FUNCTION_BLOCK FB_TimeDelta
VAR
	StartTime : ST_TimeStruct;
    StopTime : ST_TimeStruct;
    CurrentTime : ST_TimeStruct; // Assuming this to be cyclically updated to the current PLC time
	fbGetSystemTime : GETSYSTEMTIME;
    timeAsFileTime : T_FILETIME;
    timeAsDT : DATE_AND_TIME;
END_VAR

F_GetSystemTime(F_GetSystemTime => CurrentTime);
GetDelta();

METHOD GetDelta : ST_TimeStruct
VAR
	DeltaTime : ST_TimeStruct;
	DaysInMonth : ARRAY[0..12] OF WORD := [0,31,28,31,30,31,30,31,31,30,31,30,31]; // Days in each month
	bLeapYear : BOOL;
END_VAR
// Calculate the delta TIME here AND assign it TO DeltaTime
	DeltaTime.wYear := StopTime.wYear - StartTime.wYear;
    DeltaTime.wMonth := StopTime.wMonth - StartTime.wMonth;
    DeltaTime.wDay := StopTime.wDay - StartTime.wDay;
    DeltaTime.wHour := StopTime.wHour - StartTime.wHour;
    DeltaTime.wMinute := StopTime.wMinute - StartTime.wMinute;
    DeltaTime.wSecond := StopTime.wSecond - StartTime.wSecond;
    DeltaTime.wMilliseconds := StopTime.wMilliseconds - StartTime.wMilliseconds;
	
// Calculate delta time
    IF StartTime.wMilliseconds > StopTime.wMilliseconds THEN
        DeltaTime.wMilliseconds := 65535 - DeltaTime.wMilliseconds;
    END_IF;

    IF StartTime.wSecond > StopTime.wSecond  THEN
        DeltaTime.wSecond := 65535 - DeltaTime.wSecond;
    END_IF;
	
    IF StartTime.wMinute > StopTime.wMinute THEN
        DeltaTime.wMinute := 65535 - DeltaTime.wMinute;
    END_IF;

	IF StartTime.wHour > StopTime.wHour THEN
        DeltaTime.wHour := 65535 - DeltaTime.wHour;
    END_IF;

    // Adjust for overflows
    IF DeltaTime.wMilliseconds >= 1000 THEN
        DeltaTime.wMilliseconds := DeltaTime.wMilliseconds - 1000;
        DeltaTime.wSecond := DeltaTime.wSecond + 1;
    END_IF;

    IF DeltaTime.wSecond >= 60 THEN
        DeltaTime.wSecond := DeltaTime.wSecond - 60;
        DeltaTime.wMinute := DeltaTime.wMinute + 1;
    END_IF;

    IF DeltaTime.wMinute >= 60 THEN
        DeltaTime.wMinute := DeltaTime.wMinute - 60;
        DeltaTime.wHour := DeltaTime.wHour + 1;
    END_IF;

    IF DeltaTime.wHour >= 24 THEN
        DeltaTime.wHour := DeltaTime.wHour - 24;
        DeltaTime.wDay := DeltaTime.wDay + 1;
    END_IF;

    // Check for leap year
    bLeapYear := ((StartTime.wYear MOD 4 = 0) AND (StartTime.wYear MOD 100 <> 0)) OR (StartTime.wYear MOD 400 = 0);
    IF bLeapYear THEN
        DaysInMonth[2] := 29;
    ELSE
        DaysInMonth[2] := 28;
    END_IF;

    IF DeltaTime.wDay >= DaysInMonth[StartTime.wMonth] THEN
        DeltaTime.wDay := DeltaTime.wDay - DaysInMonth[StartTime.wMonth];
        DeltaTime.wMonth := DeltaTime.wMonth + 1;
    END_IF;

    IF DeltaTime.wMonth >= 12 THEN
        DeltaTime.wMonth := DeltaTime.wMonth - 12;
        DeltaTime.wYear := DeltaTime.wYear + 1;
    END_IF;

    // Return the calculated delta time
    GetDelta := DeltaTime;
END_METHOD

METHOD Start : ST_TimeStruct
VAR
END_VAR
// Assume CurrentTime is updated externally and cyclically with the current PLC time
F_GetSystemTime(F_GetSystemTime => StartTime);
END_METHOD

METHOD Stop : ST_TimeStruct
VAR
END_VAR
// Assume CurrentTime is updated externally and cyclically with the current PLC time
F_GetSystemTime(F_GetSystemTime => StopTime);
END_METHOD

END_FUNCTION_BLOCK

(* stored: Version 1.1.0.1, ProductVersion 3.1.4024.12
   POU FB_TimeDelta: Id {b5ea659c-d259-44ba-9ffb-24d656cf8516}, SpecialFunc None
   Method GetDelta: Id {dc148d7e-5e4a-4f58-9089-0c666953aba3}
   Method Start: Id {4d2d0b47-78d8-47e4-8b2c-a9bcca0370d5}
   Method Stop: Id {be9a23e9-38d7-472e-8d3c-f7f558ab2be6} *)
